// Mitsubishi GX Works2 project: b15   PLC: Q02/Q02H

PROGRAM MAIN
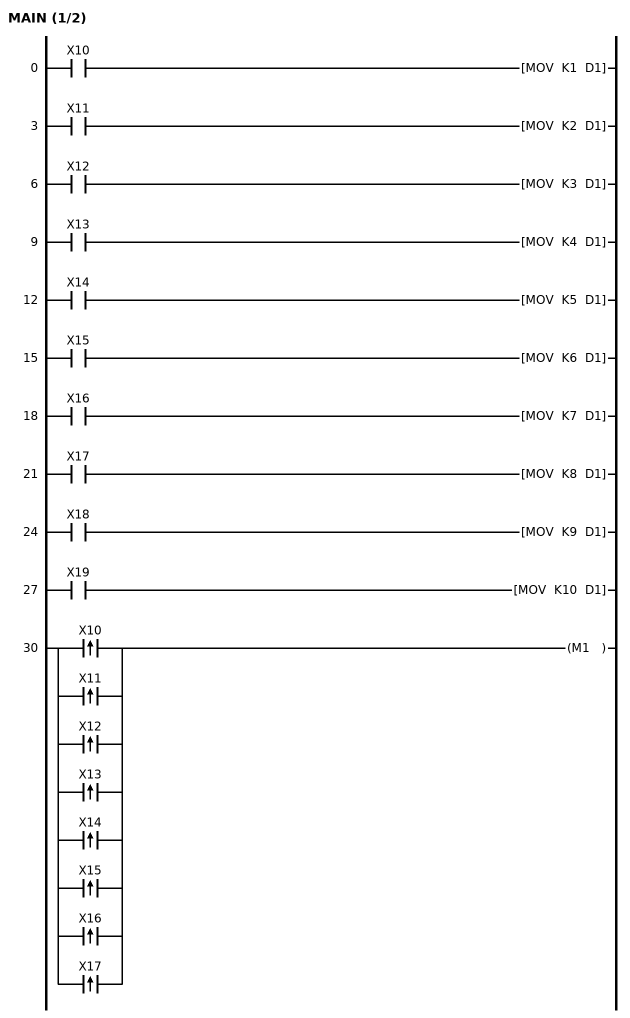
0     LD      X10
      MOV     K1 D1
3     LD      X11
      MOV     K2 D1
6     LD      X12
      MOV     K3 D1
9     LD      X13
      MOV     K4 D1
12    LD      X14
      MOV     K5 D1
15    LD      X15
      MOV     K6 D1
18    LD      X16
      MOV     K7 D1
21    LD      X17
      MOV     K8 D1
24    LD      X18
      MOV     K9 D1
27    LD      X19
      MOV     K10 D1
30    LDP     X10
      ORP     X11
      ORP     X12
      ORP     X13
      ORP     X14
      ORP     X15
      ORP     X16
      ORP     X17
      OUT     M1
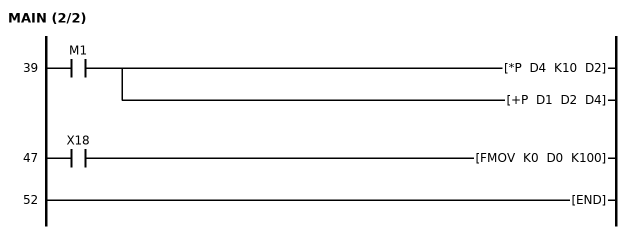
39    LD      M1
      *P      D4 K10 D2
      +P      D1 D2 D4
47    LD      X18
      FMOV    K0 D0 K100
52    END
END_PROGRAM
